(* CoDeSys 2.3 export: HandlerEkor0.EXP *)

(* POU SGL_Sismored/Sismored 4.0/New_telemetry_model/HandlerEkor0, ST *)
FUNCTION HandlerEkor0 : BOOL
VAR_INPUT
	eError : eErrorCodes;

END_VAR
VAR
	sErrorDescription : STRING;

END_VAR
IF eError <> NO_ERROR THEN
        CASE eError OF

			EXECUTION_ERROR	:	sErrorDescription := 'EXECUTION_ERROR';

			TIMEOFF_ERROR		:	sErrorDescription := 'TIMEOFF_ERROR';

			COM_ERROR			:	sErrorDescription := 'COM_ERROR';

		ELSE
			(* Unknown error *)
			sErrorDescription := 'UNKNOWN_ERROR';
		END_CASE;

	SaveError(sErrorDescription);
	HandlerEkor0 := TRUE;
END_IF
END_FUNCTION
